Staubli VAL3: PositionTrigger.pgx

program PositionTrigger()
  local num nhere
begin
  ntime=clock()
  nnnn=0
  shere=pfrmCad[0]
  call Transmission()
  delay(0)

  while true
    if bSignal==true
      //shere=here(tTool,FrmDraw)
      shere=here(tTool,world)
      fout=false
      delay(0)
      fout=true
      delay(0.005)
      call Transmission()
      delay(0)
      ndelay=clock()-ntime
      nnnn=nnnn+1
    endIf
    delay(0)

  endWhile
  ndelay=clock()-ntime
end
